(* PLC project FiveDofPlatform_v26085.modbus_registers.import.xml, CODESYS CODESYS V3.5 SP20 Patch 4 *)
(* stored: creationDateTime 2026-08-01T14:33:36, modificationDateTime 2026-08-01T14:33:36 *)

PROGRAM AxisEnableControl_PRG
  VAR
    i : INT;
    xEnableAll : BOOL;
    wEnableFeedback : WORD;
  END_VAR

            
// v26085：五轴使能寄存器 arReg_data[32] 已集中到 ModbusTcpSlave 解析。
// 本程序只保留任务调用占位，不再读写 arReg_data，避免同一个寄存器被多处写入。
          
END_PROGRAM

PROGRAM FiveDOF_Platform_PRG
  VAR
    final_angle : ARRAY[1..AXIS_COUNT] OF LREAL;  (* 最终目标 *)
    final_vel : ARRAY[1..AXIS_COUNT] OF LREAL;
    fbMove_2 : FB_5DOF_Platform_Move;  (* 功能块实例 *)
    trig_start : R_TRIG;  (* 触发边沿检测 *)
    i : INT;  (* 辅助 *)
    log_msg : STRING(255);
    logfb : Syslog_FB;
  END_VAR

            
// --------------------------------------------------
// 主逻辑
// --------------------------------------------------
// 五轴使能由 AxisEnableControl_PRG 根据 arReg_data[32] 统一控制。
// 这里不再每周期强制 TRUE，避免覆盖寄存器关闭使能命令。
// v26085：arAi_data[9] 五轴运行状态输入寄存器改由 ModbusTcpSlave 统一写出。
// 本程序只维护内部状态变量 bfiveDOF_state。
// 检测外部移动指令
trig_start(CLK := Move_5Axis_Sign=1);
IF trig_start.Q THEN

	log_msg := 'five-axis platform starts moving';
// 	logfb(write:=TRUE,sFileTestString:=log_msg);
	AppendLog(log_msg);

    // 使能所有轴（可放在这里一次性使能）
	bfiveDOF_state:=1;//开始运动
    AppendLog('status 0:6-axis start move' );
    step := 10;   // 开始安全顺序
END_IF

CASE step OF
    0: // 空闲
		bfiveDOF_state:=0;//开始运动
    // ---------- 阶段1：轴移动到目标 ----------
    10:
		FOR i := 1 TO AXIS_COUNT DO
			final_angle[i] := PlatformTargetAngle[i];
			final_vel[i]   := 360*6000/60;
			Axes[i].AxisDone := FALSE;  
			GVL.Axes[i].NeedMoveAxis := TRUE;
		END_FOR
        fbMove_2(AxisAngle := final_angle, AxisVel := final_vel, Execute := TRUE,Monitor:=TRUE);
        step := 20;

		log_msg := 'State 20: Start moving XYABC AXIS... ';
// 		logfb(write:=TRUE,sFileTestString:=log_msg);
		AppendLog(log_msg);;
    20:
        fbMove_2(AxisAngle := final_angle, AxisVel := final_vel, Execute := FALSE,Monitor:=TRUE);
        IF fbMove_2.allDone THEN
			log_msg := 'State 21: XYZABC AXIS movement completed';
// 			logfb(write:=TRUE,sFileTestString:=log_msg);
			AppendLog(log_msg);
        ELSIF fbMove_2.Error THEN
            bfiveDOF_state:=2;
        END_IF
		step := 0;

        
        
END_CASE
          
END_PROGRAM

PROGRAM AxisStatusFeedback_PRG
  VAR
    fbStatusX : Sm3_Basic.MC_ReadStatus;
    fbAxisErrorX : Sm3_Basic.MC_ReadAxisError;
    fbStatusY : Sm3_Basic.MC_ReadStatus;
    fbAxisErrorY : Sm3_Basic.MC_ReadAxisError;
    fbStatusZ : Sm3_Basic.MC_ReadStatus;
    fbAxisErrorZ : Sm3_Basic.MC_ReadAxisError;
    fbStatusB : Sm3_Basic.MC_ReadStatus;
    fbAxisErrorB : Sm3_Basic.MC_ReadAxisError;
    fbStatusC : Sm3_Basic.MC_ReadStatus;
    fbAxisErrorC : Sm3_Basic.MC_ReadAxisError;
    wStatusX : WORD;
    wStatusY : WORD;
    wStatusZ : WORD;
    wStatusB : WORD;
    wStatusC : WORD;
    dwAxisErrorX : DWORD;
    dwAxisErrorY : DWORD;
    dwAxisErrorZ : DWORD;
    dwAxisErrorB : DWORD;
    dwAxisErrorC : DWORD;
    bStatusErrorX : BOOL;
    bStatusFBErrorX : BOOL;
    bAxisErrorX : BOOL;
    bSwEndSwitchX : BOOL;
    bStatusErrorY : BOOL;
    bStatusFBErrorY : BOOL;
    bAxisErrorY : BOOL;
    bSwEndSwitchY : BOOL;
    bStatusErrorZ : BOOL;
    bStatusFBErrorZ : BOOL;
    bAxisErrorZ : BOOL;
    bSwEndSwitchZ : BOOL;
    bStatusErrorB : BOOL;
    bStatusFBErrorB : BOOL;
    bAxisErrorB : BOOL;
    bSwEndSwitchB : BOOL;
    bStatusErrorC : BOOL;
    bStatusFBErrorC : BOOL;
    bAxisErrorC : BOOL;
    bSwEndSwitchC : BOOL;
    eStatusErrorX : SMC_ERROR;
    eAxisReadErrorX : SMC_ERROR;
    bAxisReadErrorX : BOOL;
    eStatusErrorY : SMC_ERROR;
    eAxisReadErrorY : SMC_ERROR;
    bAxisReadErrorY : BOOL;
    eStatusErrorZ : SMC_ERROR;
    eAxisReadErrorZ : SMC_ERROR;
    bAxisReadErrorZ : BOOL;
    eStatusErrorB : SMC_ERROR;
    eAxisReadErrorB : SMC_ERROR;
    bAxisReadErrorB : BOOL;
    eStatusErrorC : SMC_ERROR;
    eAxisReadErrorC : SMC_ERROR;
    bAxisReadErrorC : BOOL;
    wEnableMismatchFeedback : WORD;
    wStatusErrorFeedback : WORD;
    wAxisReadErrorFeedback : WORD;
    wStatusFBErrorFeedback : WORD;
  END_VAR

            
// v26085：本程序只读取 SoftMotion 状态并写入全局缓存。
// 所有 arReg_data 寄存器地址统一在 ModbusTcpSlave 中写出，方便集中排查。

fbStatusX(
    Axis := AXIS_X,
    Enable := TRUE,
    Valid => ,
    Busy => ,
    Error => bStatusErrorX,
    ErrorID => eStatusErrorX,
    Disabled => ,
    Errorstop => ,
    Stopping => ,
    StandStill => ,
    DiscreteMotion => ,
    ContinuousMotion => ,
    SynchronizedMotion => ,
    Homing => ,
    ConstantVelocity => ,
    Accelerating => ,
    Decelerating => ,
    FBErrorOccured => bStatusFBErrorX,
);

// 读取 X 轴本体错误。这里不直接写 arReg_data，寄存器统一由 ModbusTcpSlave 输出。
fbAxisErrorX(
    Axis := AXIS_X,
    Enable := TRUE,
    Valid => ,
    Busy => ,
    Error => bAxisReadErrorX,
    ErrorID => eAxisReadErrorX,
    AxisError => bAxisErrorX,
    AxisErrorID => dwAxisErrorX,
    SWEndSwitchActive => bSwEndSwitchX
);
IF NOT bAxisErrorX THEN
    // 无轴本体错误时清零 AxisErrorID 缓存，避免保留上一次错误号。
    dwAxisErrorX := DWORD#0;
END_IF;

// 把 X 轴状态压缩成 WORD 缓存。实际 arReg_data[33] 由 ModbusTcpSlave 写出。
wStatusX := WORD#0;
IF fbStatusX.Disabled THEN wStatusX := wStatusX OR WORD#16#0001; END_IF;
IF fbStatusX.Errorstop THEN wStatusX := wStatusX OR WORD#16#0002; END_IF;
IF fbStatusX.Stopping THEN wStatusX := wStatusX OR WORD#16#0004; END_IF;
IF fbStatusX.StandStill THEN wStatusX := wStatusX OR WORD#16#0008; END_IF;
IF fbStatusX.DiscreteMotion THEN wStatusX := wStatusX OR WORD#16#0010; END_IF;
IF fbStatusX.ContinuousMotion THEN wStatusX := wStatusX OR WORD#16#0020; END_IF;
IF fbStatusX.SynchronizedMotion THEN wStatusX := wStatusX OR WORD#16#0040; END_IF;
IF fbStatusX.Homing THEN wStatusX := wStatusX OR WORD#16#0080; END_IF;
IF fbStatusX.ConstantVelocity THEN wStatusX := wStatusX OR WORD#16#0100; END_IF;
IF fbStatusX.Accelerating THEN wStatusX := wStatusX OR WORD#16#0200; END_IF;
IF fbStatusX.Decelerating THEN wStatusX := wStatusX OR WORD#16#0400; END_IF;
IF bAxisErrorX THEN wStatusX := wStatusX OR WORD#16#4000; END_IF;
IF bSwEndSwitchX THEN wStatusX := wStatusX OR WORD#16#8000; END_IF;
wAxisStatusReg[1] := wStatusX;

// 错误号先放入全局缓存，ModbusTcpSlave 统一拆成低/高 16 位寄存器。
dwAxisErrorIDReg[1] := dwAxisErrorX;
dwReadStatusErrorIDReg[1] := TO_DWORD(eStatusErrorX);
dwReadAxisErrorFBIDReg[1] := TO_DWORD(eAxisReadErrorX);

fbStatusY(
    Axis := AXIS_Y,
    Enable := TRUE,
    Valid => ,
    Busy => ,
    Error => bStatusErrorY,
    ErrorID => eStatusErrorY,
    Disabled => ,
    Errorstop => ,
    Stopping => ,
    StandStill => ,
    DiscreteMotion => ,
    ContinuousMotion => ,
    SynchronizedMotion => ,
    Homing => ,
    ConstantVelocity => ,
    Accelerating => ,
    Decelerating => ,
    FBErrorOccured => bStatusFBErrorY,
);

// 读取 Y 轴本体错误。这里不直接写 arReg_data，寄存器统一由 ModbusTcpSlave 输出。
fbAxisErrorY(
    Axis := AXIS_Y,
    Enable := TRUE,
    Valid => ,
    Busy => ,
    Error => bAxisReadErrorY,
    ErrorID => eAxisReadErrorY,
    AxisError => bAxisErrorY,
    AxisErrorID => dwAxisErrorY,
    SWEndSwitchActive => bSwEndSwitchY
);
IF NOT bAxisErrorY THEN
    // 无轴本体错误时清零 AxisErrorID 缓存，避免保留上一次错误号。
    dwAxisErrorY := DWORD#0;
END_IF;

// 把 Y 轴状态压缩成 WORD 缓存。实际 arReg_data[34] 由 ModbusTcpSlave 写出。
wStatusY := WORD#0;
IF fbStatusY.Disabled THEN wStatusY := wStatusY OR WORD#16#0001; END_IF;
IF fbStatusY.Errorstop THEN wStatusY := wStatusY OR WORD#16#0002; END_IF;
IF fbStatusY.Stopping THEN wStatusY := wStatusY OR WORD#16#0004; END_IF;
IF fbStatusY.StandStill THEN wStatusY := wStatusY OR WORD#16#0008; END_IF;
IF fbStatusY.DiscreteMotion THEN wStatusY := wStatusY OR WORD#16#0010; END_IF;
IF fbStatusY.ContinuousMotion THEN wStatusY := wStatusY OR WORD#16#0020; END_IF;
IF fbStatusY.SynchronizedMotion THEN wStatusY := wStatusY OR WORD#16#0040; END_IF;
IF fbStatusY.Homing THEN wStatusY := wStatusY OR WORD#16#0080; END_IF;
IF fbStatusY.ConstantVelocity THEN wStatusY := wStatusY OR WORD#16#0100; END_IF;
IF fbStatusY.Accelerating THEN wStatusY := wStatusY OR WORD#16#0200; END_IF;
IF fbStatusY.Decelerating THEN wStatusY := wStatusY OR WORD#16#0400; END_IF;
IF bAxisErrorY THEN wStatusY := wStatusY OR WORD#16#4000; END_IF;
IF bSwEndSwitchY THEN wStatusY := wStatusY OR WORD#16#8000; END_IF;
wAxisStatusReg[2] := wStatusY;

// 错误号先放入全局缓存，ModbusTcpSlave 统一拆成低/高 16 位寄存器。
dwAxisErrorIDReg[2] := dwAxisErrorY;
dwReadStatusErrorIDReg[2] := TO_DWORD(eStatusErrorY);
dwReadAxisErrorFBIDReg[2] := TO_DWORD(eAxisReadErrorY);

fbStatusZ(
    Axis := AXIS_Z,
    Enable := TRUE,
    Valid => ,
    Busy => ,
    Error => bStatusErrorZ,
    ErrorID => eStatusErrorZ,
    Disabled => ,
    Errorstop => ,
    Stopping => ,
    StandStill => ,
    DiscreteMotion => ,
    ContinuousMotion => ,
    SynchronizedMotion => ,
    Homing => ,
    ConstantVelocity => ,
    Accelerating => ,
    Decelerating => ,
    FBErrorOccured => bStatusFBErrorZ,
);

// 读取 Z 轴本体错误。这里不直接写 arReg_data，寄存器统一由 ModbusTcpSlave 输出。
fbAxisErrorZ(
    Axis := AXIS_Z,
    Enable := TRUE,
    Valid => ,
    Busy => ,
    Error => bAxisReadErrorZ,
    ErrorID => eAxisReadErrorZ,
    AxisError => bAxisErrorZ,
    AxisErrorID => dwAxisErrorZ,
    SWEndSwitchActive => bSwEndSwitchZ
);
IF NOT bAxisErrorZ THEN
    // 无轴本体错误时清零 AxisErrorID 缓存，避免保留上一次错误号。
    dwAxisErrorZ := DWORD#0;
END_IF;

// 把 Z 轴状态压缩成 WORD 缓存。实际 arReg_data[35] 由 ModbusTcpSlave 写出。
wStatusZ := WORD#0;
IF fbStatusZ.Disabled THEN wStatusZ := wStatusZ OR WORD#16#0001; END_IF;
IF fbStatusZ.Errorstop THEN wStatusZ := wStatusZ OR WORD#16#0002; END_IF;
IF fbStatusZ.Stopping THEN wStatusZ := wStatusZ OR WORD#16#0004; END_IF;
IF fbStatusZ.StandStill THEN wStatusZ := wStatusZ OR WORD#16#0008; END_IF;
IF fbStatusZ.DiscreteMotion THEN wStatusZ := wStatusZ OR WORD#16#0010; END_IF;
IF fbStatusZ.ContinuousMotion THEN wStatusZ := wStatusZ OR WORD#16#0020; END_IF;
IF fbStatusZ.SynchronizedMotion THEN wStatusZ := wStatusZ OR WORD#16#0040; END_IF;
IF fbStatusZ.Homing THEN wStatusZ := wStatusZ OR WORD#16#0080; END_IF;
IF fbStatusZ.ConstantVelocity THEN wStatusZ := wStatusZ OR WORD#16#0100; END_IF;
IF fbStatusZ.Accelerating THEN wStatusZ := wStatusZ OR WORD#16#0200; END_IF;
IF fbStatusZ.Decelerating THEN wStatusZ := wStatusZ OR WORD#16#0400; END_IF;
IF bAxisErrorZ THEN wStatusZ := wStatusZ OR WORD#16#4000; END_IF;
IF bSwEndSwitchZ THEN wStatusZ := wStatusZ OR WORD#16#8000; END_IF;
wAxisStatusReg[3] := wStatusZ;

// 错误号先放入全局缓存，ModbusTcpSlave 统一拆成低/高 16 位寄存器。
dwAxisErrorIDReg[3] := dwAxisErrorZ;
dwReadStatusErrorIDReg[3] := TO_DWORD(eStatusErrorZ);
dwReadAxisErrorFBIDReg[3] := TO_DWORD(eAxisReadErrorZ);

fbStatusB(
    Axis := AXIS_B,
    Enable := TRUE,
    Valid => ,
    Busy => ,
    Error => bStatusErrorB,
    ErrorID => eStatusErrorB,
    Disabled => ,
    Errorstop => ,
    Stopping => ,
    StandStill => ,
    DiscreteMotion => ,
    ContinuousMotion => ,
    SynchronizedMotion => ,
    Homing => ,
    ConstantVelocity => ,
    Accelerating => ,
    Decelerating => ,
    FBErrorOccured => bStatusFBErrorB,
);

// 读取 B 轴本体错误。这里不直接写 arReg_data，寄存器统一由 ModbusTcpSlave 输出。
fbAxisErrorB(
    Axis := AXIS_B,
    Enable := TRUE,
    Valid => ,
    Busy => ,
    Error => bAxisReadErrorB,
    ErrorID => eAxisReadErrorB,
    AxisError => bAxisErrorB,
    AxisErrorID => dwAxisErrorB,
    SWEndSwitchActive => bSwEndSwitchB
);
IF NOT bAxisErrorB THEN
    // 无轴本体错误时清零 AxisErrorID 缓存，避免保留上一次错误号。
    dwAxisErrorB := DWORD#0;
END_IF;

// 把 B 轴状态压缩成 WORD 缓存。实际 arReg_data[36] 由 ModbusTcpSlave 写出。
wStatusB := WORD#0;
IF fbStatusB.Disabled THEN wStatusB := wStatusB OR WORD#16#0001; END_IF;
IF fbStatusB.Errorstop THEN wStatusB := wStatusB OR WORD#16#0002; END_IF;
IF fbStatusB.Stopping THEN wStatusB := wStatusB OR WORD#16#0004; END_IF;
IF fbStatusB.StandStill THEN wStatusB := wStatusB OR WORD#16#0008; END_IF;
IF fbStatusB.DiscreteMotion THEN wStatusB := wStatusB OR WORD#16#0010; END_IF;
IF fbStatusB.ContinuousMotion THEN wStatusB := wStatusB OR WORD#16#0020; END_IF;
IF fbStatusB.SynchronizedMotion THEN wStatusB := wStatusB OR WORD#16#0040; END_IF;
IF fbStatusB.Homing THEN wStatusB := wStatusB OR WORD#16#0080; END_IF;
IF fbStatusB.ConstantVelocity THEN wStatusB := wStatusB OR WORD#16#0100; END_IF;
IF fbStatusB.Accelerating THEN wStatusB := wStatusB OR WORD#16#0200; END_IF;
IF fbStatusB.Decelerating THEN wStatusB := wStatusB OR WORD#16#0400; END_IF;
IF bAxisErrorB THEN wStatusB := wStatusB OR WORD#16#4000; END_IF;
IF bSwEndSwitchB THEN wStatusB := wStatusB OR WORD#16#8000; END_IF;
wAxisStatusReg[4] := wStatusB;

// 错误号先放入全局缓存，ModbusTcpSlave 统一拆成低/高 16 位寄存器。
dwAxisErrorIDReg[4] := dwAxisErrorB;
dwReadStatusErrorIDReg[4] := TO_DWORD(eStatusErrorB);
dwReadAxisErrorFBIDReg[4] := TO_DWORD(eAxisReadErrorB);

fbStatusC(
    Axis := AXIS_C,
    Enable := TRUE,
    Valid => ,
    Busy => ,
    Error => bStatusErrorC,
    ErrorID => eStatusErrorC,
    Disabled => ,
    Errorstop => ,
    Stopping => ,
    StandStill => ,
    DiscreteMotion => ,
    ContinuousMotion => ,
    SynchronizedMotion => ,
    Homing => ,
    ConstantVelocity => ,
    Accelerating => ,
    Decelerating => ,
    FBErrorOccured => bStatusFBErrorC,
);

// 读取 C 轴本体错误。这里不直接写 arReg_data，寄存器统一由 ModbusTcpSlave 输出。
fbAxisErrorC(
    Axis := AXIS_C,
    Enable := TRUE,
    Valid => ,
    Busy => ,
    Error => bAxisReadErrorC,
    ErrorID => eAxisReadErrorC,
    AxisError => bAxisErrorC,
    AxisErrorID => dwAxisErrorC,
    SWEndSwitchActive => bSwEndSwitchC
);
IF NOT bAxisErrorC THEN
    // 无轴本体错误时清零 AxisErrorID 缓存，避免保留上一次错误号。
    dwAxisErrorC := DWORD#0;
END_IF;

// 把 C 轴状态压缩成 WORD 缓存。实际 arReg_data[37] 由 ModbusTcpSlave 写出。
wStatusC := WORD#0;
IF fbStatusC.Disabled THEN wStatusC := wStatusC OR WORD#16#0001; END_IF;
IF fbStatusC.Errorstop THEN wStatusC := wStatusC OR WORD#16#0002; END_IF;
IF fbStatusC.Stopping THEN wStatusC := wStatusC OR WORD#16#0004; END_IF;
IF fbStatusC.StandStill THEN wStatusC := wStatusC OR WORD#16#0008; END_IF;
IF fbStatusC.DiscreteMotion THEN wStatusC := wStatusC OR WORD#16#0010; END_IF;
IF fbStatusC.ContinuousMotion THEN wStatusC := wStatusC OR WORD#16#0020; END_IF;
IF fbStatusC.SynchronizedMotion THEN wStatusC := wStatusC OR WORD#16#0040; END_IF;
IF fbStatusC.Homing THEN wStatusC := wStatusC OR WORD#16#0080; END_IF;
IF fbStatusC.ConstantVelocity THEN wStatusC := wStatusC OR WORD#16#0100; END_IF;
IF fbStatusC.Accelerating THEN wStatusC := wStatusC OR WORD#16#0200; END_IF;
IF fbStatusC.Decelerating THEN wStatusC := wStatusC OR WORD#16#0400; END_IF;
IF bAxisErrorC THEN wStatusC := wStatusC OR WORD#16#4000; END_IF;
IF bSwEndSwitchC THEN wStatusC := wStatusC OR WORD#16#8000; END_IF;
wAxisStatusReg[5] := wStatusC;

// 错误号先放入全局缓存，ModbusTcpSlave 统一拆成低/高 16 位寄存器。
dwAxisErrorIDReg[5] := dwAxisErrorC;
dwReadStatusErrorIDReg[5] := TO_DWORD(eStatusErrorC);
dwReadAxisErrorFBIDReg[5] := TO_DWORD(eAxisReadErrorC);

// 使能请求不一致：AxisEnable 请求 TRUE，但轴状态仍 Disabled。
wEnableMismatchFeedback := WORD#0;
IF GVL.Axes[1].AxisEnable AND fbStatusX.Disabled THEN wEnableMismatchFeedback := wEnableMismatchFeedback OR WORD#16#0001; END_IF;
IF GVL.Axes[2].AxisEnable AND fbStatusY.Disabled THEN wEnableMismatchFeedback := wEnableMismatchFeedback OR WORD#16#0002; END_IF;
IF GVL.Axes[3].AxisEnable AND fbStatusZ.Disabled THEN wEnableMismatchFeedback := wEnableMismatchFeedback OR WORD#16#0004; END_IF;
IF GVL.Axes[4].AxisEnable AND fbStatusB.Disabled THEN wEnableMismatchFeedback := wEnableMismatchFeedback OR WORD#16#0008; END_IF;
IF GVL.Axes[5].AxisEnable AND fbStatusC.Disabled THEN wEnableMismatchFeedback := wEnableMismatchFeedback OR WORD#16#0010; END_IF;
wEnableMismatchReg := wEnableMismatchFeedback;

// MC_ReadStatus.Error 汇总位，bit0..bit4=X/Y/Z/B/C。
wStatusErrorFeedback := WORD#0;
IF bStatusErrorX THEN wStatusErrorFeedback := wStatusErrorFeedback OR WORD#16#0001; END_IF;
IF bStatusErrorY THEN wStatusErrorFeedback := wStatusErrorFeedback OR WORD#16#0002; END_IF;
IF bStatusErrorZ THEN wStatusErrorFeedback := wStatusErrorFeedback OR WORD#16#0004; END_IF;
IF bStatusErrorB THEN wStatusErrorFeedback := wStatusErrorFeedback OR WORD#16#0008; END_IF;
IF bStatusErrorC THEN wStatusErrorFeedback := wStatusErrorFeedback OR WORD#16#0010; END_IF;
wReadStatusErrorBitsReg := wStatusErrorFeedback;

// MC_ReadAxisError.Error 汇总位，bit0..bit4=X/Y/Z/B/C。
wAxisReadErrorFeedback := WORD#0;
IF bAxisReadErrorX THEN wAxisReadErrorFeedback := wAxisReadErrorFeedback OR WORD#16#0001; END_IF;
IF bAxisReadErrorY THEN wAxisReadErrorFeedback := wAxisReadErrorFeedback OR WORD#16#0002; END_IF;
IF bAxisReadErrorZ THEN wAxisReadErrorFeedback := wAxisReadErrorFeedback OR WORD#16#0004; END_IF;
IF bAxisReadErrorB THEN wAxisReadErrorFeedback := wAxisReadErrorFeedback OR WORD#16#0008; END_IF;
IF bAxisReadErrorC THEN wAxisReadErrorFeedback := wAxisReadErrorFeedback OR WORD#16#0010; END_IF;
wReadAxisErrorBitsReg := wAxisReadErrorFeedback;

// MC_ReadStatus.FBErrorOccured 汇总位，bit0..bit4=X/Y/Z/B/C。
wStatusFBErrorFeedback := WORD#0;
IF bStatusFBErrorX THEN wStatusFBErrorFeedback := wStatusFBErrorFeedback OR WORD#16#0001; END_IF;
IF bStatusFBErrorY THEN wStatusFBErrorFeedback := wStatusFBErrorFeedback OR WORD#16#0002; END_IF;
IF bStatusFBErrorZ THEN wStatusFBErrorFeedback := wStatusFBErrorFeedback OR WORD#16#0004; END_IF;
IF bStatusFBErrorB THEN wStatusFBErrorFeedback := wStatusFBErrorFeedback OR WORD#16#0008; END_IF;
IF bStatusFBErrorC THEN wStatusFBErrorFeedback := wStatusFBErrorFeedback OR WORD#16#0010; END_IF;
wReadStatusFBErrorBitsReg := wStatusFBErrorFeedback;

          
END_PROGRAM

PROGRAM AXIS_X_PRG
  VAR
    伺服使能 : Sm3_Basic.MC_Power;  (* 轴功能块实例 *)
    伺服绝对位置执行 : Sm3_Basic.MC_MoveAbsolute;
    伺服实际位置 : Sm3_Basic.MC_ReadActualPosition;
    伺服停止 : Sm3_Basic.MC_Stop;
    伺服复位 : Sm3_Basic.MC_Reset;
    伺服状态 : Sm3_Basic.MC_ReadStatus;
    复位轴组 : Sm3_Basic.SMC3_ReinitDrive;
    当前位置 : LREAL;  (* 变量 *)
    轴组复位 : BOOL;
    目标位置 : LREAL;
    目标速度 : LREAL;
    伺服错误状态 : BOOL;
    轴使能状态 : BOOL;
    总线状态 : BOOL;
    复位触发 : R_TRIG;  (* 报警清除相关 *)
    复位请求 : BOOL;
    复位中 : BOOL;
    POS_DEAD_ZONE : REAL := 0.01;  (* 死区常量 *)
    move_trigger : R_TRIG;
    AXIS_X_EXCUSE : BOOL := FALSE;
    log_msg : STRING(100);
    bPowerErrorDiag : BOOL;
    ePowerErrorDiag : SMC_ERROR;
    wPowerDiag : WORD;
  END_VAR

            //------------------------------------------------------------------
// Z 轴控制逻辑（简化版 - 仅上升沿触发）
//------------------------------------------------------------------

// 读取实际位置
伺服实际位置(
    Axis    := AXIS_X,
    Enable  := TRUE,
    Position=> 当前位置
);
GVL.Axes[1].ActualAngle := 当前位置;

// 读取轴状态
伺服状态(
    Axis    := AXIS_X,
    Enable  := TRUE,
    Valid   => ,
    Busy    => ,
    Error   => 伺服错误状态,
    ErrorID => ,
    Disabled=> 总线状态
);

// 轴使能控制
伺服使能(
    Axis               := AXIS_X,
    Enable             := TRUE,
    bRegulatorOn       := GVL.Axes[1].AxisEnable,
    bDriveStart        := GVL.Axes[1].AxisEnable,
    Status             => 轴使能状态,
    bRegulatorRealState=> ,
    bDriveStartRealState=> ,
    Busy               => ,
    Error              => bPowerErrorDiag,
    ErrorID            => ePowerErrorDiag
);



// v26085：本轴 MC_Power 诊断先写入全局缓存，实际寄存器输出统一由 ModbusTcpSlave 完成。
dwPowerErrorIDReg[1] := TO_DWORD(ePowerErrorDiag);

// wPowerDiagReg[1] bit0=MC_Power.Status，bit1=MC_Power.Error。
wPowerDiag := WORD#0;
IF 轴使能状态 THEN wPowerDiag := wPowerDiag OR WORD#16#0001; END_IF;
IF bPowerErrorDiag THEN wPowerDiag := wPowerDiag OR WORD#16#0002; END_IF;
wPowerDiagReg[1] := wPowerDiag;

// 目标位置、速度赋值（来自全局变量）
目标位置 := GVL.Axes[1].TargetAngle;
目标速度 :=  GVL.Axes[1].TargetVel;

// ********** 核心：上升沿触发运动 **********
// 使用 R_TRIG 检测 need_move 的上升沿
move_trigger(CLK := GVL.Axes[1].NeedMoveAxis);
IF move_trigger.Q THEN
    AXIS_X_EXCUSE := TRUE;   // 产生一个扫描周期的脉冲
	log_msg := 'X-axis has been triggered';
// 	logfb(write:=TRUE,sFileTestString:=log_msg);
	AppendLog(log_msg);
ELSE
    AXIS_X_EXCUSE := FALSE;
END_IF

// 绝对定位指令
GVL.Axes[1].伺服绝对位置执行(
    Axis        := AXIS_X,
    Execute     := AXIS_X_EXCUSE,
    Position    := 目标位置,
    Velocity    := 目标速度,
    Acceleration:= 10000,//4000  //85000
    Deceleration:= 10000,//4000  //85000
    Jerk        := ,
    Direction   := ,
    BufferMode  := ,
    Done        => GVL.Axes[1].InitDone,
    Busy        => ,
    Active      => ,
    CommandAborted=> ,
    Error       => GVL.Axes[1].AxisError,
    ErrorID     =>
);

// 运动完成：清除 need_move 并通知状态机
IF  GVL.Axes[1].InitDone THEN
    GVL.Axes[1].NeedMoveAxis := FALSE;              // 清除运动请求
    GVL.Axes[1].AxisDone := TRUE;         // 通知状态机运动完成
	log_msg := 'X-Axis movement completed! ';
// 	logfb(write:=TRUE,sFileTestString:=log_msg);
// 	AppendLog(log_msg);
END_IF

// 复位功能块（保持不变）
伺服复位(
    Axis    := AXIS_X,
    Execute := 复位中 AND NOT 伺服复位.Done,
    Done    => ,
    Busy    => ,
    Error   => ,
    ErrorID =>
);

复位轴组(
    Axis      := AXIS_X,
    bExecute  := 伺服复位.Done,
    bVirtual  := FALSE,
    bDone     => ,
    bBusy     => ,
    bError    => ,
    nErrorID  =>
);

// 报警清除逻辑
复位触发(CLK := (伺服错误状态 OR 复位请求) AND NOT 复位中);
IF 复位触发.Q THEN
    复位中 := TRUE;
    复位请求 := FALSE;
END_IF

IF 伺服复位.Done THEN
    复位中 := FALSE;
END_IF
          
END_PROGRAM

PROGRAM Axis_Y_PRG
  VAR
    伺服使能 : Sm3_Basic.MC_Power;  (* 轴功能块实例 *)
    伺服绝对位置执行 : Sm3_Basic.MC_MoveAbsolute;
    伺服实际位置 : Sm3_Basic.MC_ReadActualPosition;
    伺服停止 : Sm3_Basic.MC_Stop;
    伺服复位 : Sm3_Basic.MC_Reset;
    伺服状态 : Sm3_Basic.MC_ReadStatus;
    复位轴组 : Sm3_Basic.SMC3_ReinitDrive;
    当前位置 : LREAL;  (* 变量 *)
    轴组复位 : BOOL;
    目标位置 : LREAL;
    目标速度 : LREAL;
    伺服错误状态 : BOOL;
    轴使能状态 : BOOL;
    总线状态 : BOOL;
    复位触发 : R_TRIG;  (* 报警清除相关 *)
    复位请求 : BOOL;
    复位中 : BOOL;
    POS_DEAD_ZONE : REAL := 0.01;  (* 死区常量 *)
    伺服复位_Done : BOOL;
    debug_Done_Status : BOOL;  (* 在 AXIS_Y0_PRG 中添加 *)
    debug_KeepEnable : BOOL;
    move_trigger : R_TRIG;  (* 脉冲触发相关 *)
    AXIS_Y_EXCUSE : BOOL := FALSE;
    log_msg : STRING(100);
    bPowerErrorDiag : BOOL;
    ePowerErrorDiag : SMC_ERROR;
    wPowerDiag : WORD;
  END_VAR

            //------------------------------------------------------------------
// Z 轴控制逻辑（简化版 - 仅上升沿触发）
//------------------------------------------------------------------

// 读取实际位置
伺服实际位置(
    Axis    := AXIS_Y,
    Enable  := TRUE,
    Position=> 当前位置
);
GVL.Axes[2].ActualAngle := 当前位置;

// 读取轴状态
伺服状态(
    Axis    := AXIS_Y,
    Enable  := TRUE,
    Valid   => ,
    Busy    => ,
    Error   => 伺服错误状态,
    ErrorID => ,
    Disabled=> 总线状态
);

// 轴使能控制
伺服使能(
    Axis               := AXIS_Y,
    Enable             := TRUE,
    bRegulatorOn       := GVL.Axes[2].AxisEnable,
    bDriveStart        := GVL.Axes[2].AxisEnable,
    Status             => 轴使能状态,
    bRegulatorRealState=> ,
    bDriveStartRealState=> ,
    Busy               => ,
    Error              => bPowerErrorDiag,
    ErrorID            => ePowerErrorDiag
);



// v26085：本轴 MC_Power 诊断先写入全局缓存，实际寄存器输出统一由 ModbusTcpSlave 完成。
dwPowerErrorIDReg[2] := TO_DWORD(ePowerErrorDiag);

// wPowerDiagReg[2] bit0=MC_Power.Status，bit1=MC_Power.Error。
wPowerDiag := WORD#0;
IF 轴使能状态 THEN wPowerDiag := wPowerDiag OR WORD#16#0001; END_IF;
IF bPowerErrorDiag THEN wPowerDiag := wPowerDiag OR WORD#16#0002; END_IF;
wPowerDiagReg[2] := wPowerDiag;

// 目标位置、速度赋值（来自全局变量）
目标位置 := GVL.Axes[2].TargetAngle;
目标速度 :=  GVL.Axes[2].TargetVel;

// ********** 核心：上升沿触发运动 **********
// 使用 R_TRIG 检测 need_move 的上升沿
move_trigger(CLK := GVL.Axes[2].NeedMoveAxis);
IF move_trigger.Q THEN
    AXIS_Y_EXCUSE := TRUE;   // 产生一个扫描周期的脉冲
	log_msg := 'X-axis has been triggered';
// 	logfb(write:=TRUE,sFileTestString:=log_msg);
	AppendLog(log_msg);
ELSE
    AXIS_Y_EXCUSE := FALSE;
END_IF

// 绝对定位指令
GVL.Axes[2].伺服绝对位置执行(
    Axis        := AXIS_Y,
    Execute     := AXIS_Y_EXCUSE,
    Position    := 目标位置,
    Velocity    := 目标速度,
    Acceleration:= 10000,//4000  //85000
    Deceleration:= 10000,//4000  //85000
    Jerk        := ,
    Direction   := ,
    BufferMode  := ,
    Done        => GVL.Axes[2].InitDone,
    Busy        => ,
    Active      => ,
    CommandAborted=> ,
    Error       => GVL.Axes[2].AxisError,
    ErrorID     =>
);

// 运动完成：清除 need_move 并通知状态机
IF  GVL.Axes[2].InitDone THEN
    GVL.Axes[2].NeedMoveAxis := FALSE;              // 清除运动请求
    GVL.Axes[2].AxisDone := TRUE;         // 通知状态机运动完成
	log_msg := 'X-Axis movement completed! ';
// 	logfb(write:=TRUE,sFileTestString:=log_msg);
// 	AppendLog(log_msg);
END_IF

// 复位功能块（保持不变）
伺服复位(
    Axis    := AXIS_Y,
    Execute := 复位中 AND NOT 伺服复位.Done,
    Done    => ,
    Busy    => ,
    Error   => ,
    ErrorID =>
);

复位轴组(
    Axis      := AXIS_Y,
    bExecute  := 伺服复位.Done,
    bVirtual  := FALSE,
    bDone     => ,
    bBusy     => ,
    bError    => ,
    nErrorID  =>
);

// 报警清除逻辑
复位触发(CLK := (伺服错误状态 OR 复位请求) AND NOT 复位中);
IF 复位触发.Q THEN
    复位中 := TRUE;
    复位请求 := FALSE;
END_IF

IF 伺服复位.Done THEN
    复位中 := FALSE;
END_IF
          
END_PROGRAM

PROGRAM AXIS_Z_PRG
  VAR
    伺服使能 : Sm3_Basic.MC_Power;  (* 轴功能块实例 *)
    伺服绝对位置执行 : Sm3_Basic.MC_MoveAbsolute;
    伺服实际位置 : Sm3_Basic.MC_ReadActualPosition;
    伺服停止 : Sm3_Basic.MC_Stop;
    伺服复位 : Sm3_Basic.MC_Reset;
    伺服状态 : Sm3_Basic.MC_ReadStatus;
    复位轴组 : Sm3_Basic.SMC3_ReinitDrive;
    当前位置 : LREAL;  (* 变量 *)
    轴组复位 : BOOL;
    目标位置 : LREAL;
    目标速度 : LREAL;
    伺服错误状态 : BOOL;
    轴使能状态 : BOOL;
    总线状态 : BOOL;
    复位触发 : R_TRIG;  (* 报警清除相关 *)
    复位请求 : BOOL;
    复位中 : BOOL;
    伺服复位_Done : BOOL;
    debug_Done_Status : BOOL;  (* 在 AXIS_Z_PRG 中添加 *)
    debug_KeepEnable : BOOL;
    move_trigger : R_TRIG;  (* 脉冲触发相关 *)
    AXIS_Z_EXCUSE : BOOL := FALSE;
    log_msg : STRING(100);
    bPowerErrorDiag : BOOL;
    ePowerErrorDiag : SMC_ERROR;
    wPowerDiag : WORD;
  END_VAR

            //------------------------------------------------------------------
// Z 轴控制逻辑（简化版 - 仅上升沿触发）
//------------------------------------------------------------------

// 读取实际位置
伺服实际位置(
    Axis    := AXIS_Z,
    Enable  := TRUE,
    Position=> 当前位置
);
GVL.Axes[3].ActualAngle := 当前位置;

// 读取轴状态
伺服状态(
    Axis    := AXIS_Z,
    Enable  := TRUE,
    Valid   => ,
    Busy    => ,
    Error   => 伺服错误状态,
    ErrorID => ,
    Disabled=> 总线状态
);

// 轴使能控制
伺服使能(
    Axis               := AXIS_Z,
    Enable             := TRUE,
    bRegulatorOn       := GVL.Axes[3].AxisEnable,
    bDriveStart        := GVL.Axes[3].AxisEnable,
    Status             => 轴使能状态,
    bRegulatorRealState=> ,
    bDriveStartRealState=> ,
    Busy               => ,
    Error              => bPowerErrorDiag,
    ErrorID            => ePowerErrorDiag
);



// v26085：本轴 MC_Power 诊断先写入全局缓存，实际寄存器输出统一由 ModbusTcpSlave 完成。
dwPowerErrorIDReg[3] := TO_DWORD(ePowerErrorDiag);

// wPowerDiagReg[3] bit0=MC_Power.Status，bit1=MC_Power.Error。
wPowerDiag := WORD#0;
IF 轴使能状态 THEN wPowerDiag := wPowerDiag OR WORD#16#0001; END_IF;
IF bPowerErrorDiag THEN wPowerDiag := wPowerDiag OR WORD#16#0002; END_IF;
wPowerDiagReg[3] := wPowerDiag;

// 目标位置、速度赋值（来自全局变量）
目标位置 := GVL.Axes[3].TargetAngle;
目标速度 :=  GVL.Axes[3].TargetVel;

// ********** 核心：上升沿触发运动 **********
// 使用 R_TRIG 检测 need_move 的上升沿
move_trigger(CLK := GVL.Axes[3].NeedMoveAxis);
IF move_trigger.Q THEN
    AXIS_Z_EXCUSE := TRUE;   // 产生一个扫描周期的脉冲
	log_msg := 'X-axis has been triggered';
// 	logfb(write:=TRUE,sFileTestString:=log_msg);
	AppendLog(log_msg);
ELSE
    AXIS_Z_EXCUSE := FALSE;
END_IF

// 绝对定位指令
GVL.Axes[3].伺服绝对位置执行(
    Axis        := AXIS_Z,
    Execute     := AXIS_Z_EXCUSE,
    Position    := 目标位置,
    Velocity    := 目标速度,
    Acceleration:= 10000,//4000  //85000
    Deceleration:= 10000,//4000  //85000
    Jerk        := ,
    Direction   := ,
    BufferMode  := ,
    Done        => GVL.Axes[3].InitDone,
    Busy        => ,
    Active      => ,
    CommandAborted=> ,
    Error       => GVL.Axes[3].AxisError,
    ErrorID     =>
);

// 运动完成：清除 need_move 并通知状态机
IF  GVL.Axes[3].InitDone THEN
    GVL.Axes[3].NeedMoveAxis := FALSE;              // 清除运动请求
    GVL.Axes[3].AxisDone := TRUE;         // 通知状态机运动完成
	log_msg := 'Z-Axis movement completed! ';
// 	logfb(write:=TRUE,sFileTestString:=log_msg);
// 	AppendLog(log_msg);
END_IF

// 复位功能块（保持不变）
伺服复位(
    Axis    := AXIS_Z,
    Execute := 复位中 AND NOT 伺服复位.Done,
    Done    => ,
    Busy    => ,
    Error   => ,
    ErrorID =>
);

复位轴组(
    Axis      := AXIS_Z,
    bExecute  := 伺服复位.Done,
    bVirtual  := FALSE,
    bDone     => ,
    bBusy     => ,
    bError    => ,
    nErrorID  =>
);

// 报警清除逻辑
复位触发(CLK := (伺服错误状态 OR 复位请求) AND NOT 复位中);
IF 复位触发.Q THEN
    复位中 := TRUE;
    复位请求 := FALSE;
END_IF

IF 伺服复位.Done THEN
    复位中 := FALSE;
END_IF
          
END_PROGRAM

PROGRAM AXIS_B_PRG
  VAR
    伺服使能 : Sm3_Basic.MC_Power;  (* 轴功能块实例 *)
    伺服绝对位置执行 : Sm3_Basic.MC_MoveAbsolute;
    伺服实际位置 : Sm3_Basic.MC_ReadActualPosition;
    伺服停止 : Sm3_Basic.MC_Stop;
    伺服复位 : Sm3_Basic.MC_Reset;
    伺服状态 : Sm3_Basic.MC_ReadStatus;
    复位轴组 : Sm3_Basic.SMC3_ReinitDrive;
    当前位置 : LREAL;  (* 变量 *)
    轴组复位 : BOOL;
    目标位置 : LREAL;
    目标速度 : LREAL;
    伺服错误状态 : BOOL;
    轴使能状态 : BOOL;
    总线状态 : BOOL;
    复位触发 : R_TRIG;  (* 报警清除相关 *)
    复位请求 : BOOL;
    复位中 : BOOL;
    move_trigger : R_TRIG;
    AXIS_B_EXCUSE : BOOL := FALSE;
    log_msg : STRING(100);
    bPowerErrorDiag : BOOL;
    ePowerErrorDiag : SMC_ERROR;
    wPowerDiag : WORD;
  END_VAR

            //------------------------------------------------------------------
// Z 轴控制逻辑（简化版 - 仅上升沿触发）
//------------------------------------------------------------------

// 读取实际位置
伺服实际位置(
    Axis    := AXIS_B,
    Enable  := TRUE,
    Position=> 当前位置
);
GVL.Axes[4].ActualAngle := 当前位置;

// 读取轴状态
伺服状态(
    Axis    := AXIS_B,
    Enable  := TRUE,
    Valid   => ,
    Busy    => ,
    Error   => 伺服错误状态,
    ErrorID => ,
    Disabled=> 总线状态
);

// 轴使能控制
伺服使能(
    Axis               := AXIS_B,
    Enable             := TRUE,
    bRegulatorOn       := GVL.Axes[4].AxisEnable,
    bDriveStart        := GVL.Axes[4].AxisEnable,
    Status             => 轴使能状态,
    bRegulatorRealState=> ,
    bDriveStartRealState=> ,
    Busy               => ,
    Error              => bPowerErrorDiag,
    ErrorID            => ePowerErrorDiag
);



// v26085：本轴 MC_Power 诊断先写入全局缓存，实际寄存器输出统一由 ModbusTcpSlave 完成。
dwPowerErrorIDReg[4] := TO_DWORD(ePowerErrorDiag);

// wPowerDiagReg[4] bit0=MC_Power.Status，bit1=MC_Power.Error。
wPowerDiag := WORD#0;
IF 轴使能状态 THEN wPowerDiag := wPowerDiag OR WORD#16#0001; END_IF;
IF bPowerErrorDiag THEN wPowerDiag := wPowerDiag OR WORD#16#0002; END_IF;
wPowerDiagReg[4] := wPowerDiag;

// 目标位置、速度赋值（来自全局变量）
目标位置 := GVL.Axes[4].TargetAngle;
目标速度 :=  GVL.Axes[4].TargetVel;

// ********** 核心：上升沿触发运动 **********
// 使用 R_TRIG 检测 need_move 的上升沿
move_trigger(CLK := GVL.Axes[4].NeedMoveAxis);
IF move_trigger.Q THEN
    AXIS_B_EXCUSE := TRUE;   // 产生一个扫描周期的脉冲
	log_msg := 'X-axis has been triggered';
// 	logfb(write:=TRUE,sFileTestString:=log_msg);
	AppendLog(log_msg);
ELSE
    AXIS_B_EXCUSE := FALSE;
END_IF

// 绝对定位指令
GVL.Axes[4].伺服绝对位置执行(
    Axis        := AXIS_B,
    Execute     := AXIS_B_EXCUSE,
    Position    := 目标位置,
    Velocity    := 目标速度,
    Acceleration:= 10000,//4000  //85000
    Deceleration:= 10000,//4000  //85000
    Jerk        := ,
    Direction   := ,
    BufferMode  := ,
    Done        => GVL.Axes[4].InitDone,
    Busy        => ,
    Active      => ,
    CommandAborted=> ,
    Error       => GVL.Axes[4].AxisError,
    ErrorID     =>
);

// 运动完成：清除 need_move 并通知状态机
IF  GVL.Axes[4].InitDone THEN
    GVL.Axes[4].NeedMoveAxis := FALSE;              // 清除运动请求
    GVL.Axes[4].AxisDone := TRUE;         // 通知状态机运动完成
	log_msg := 'B-Axis movement completed! ';
// 	logfb(write:=TRUE,sFileTestString:=log_msg);
// 	AppendLog(log_msg);
END_IF

// 复位功能块（保持不变）
伺服复位(
    Axis    := AXIS_B,
    Execute := 复位中 AND NOT 伺服复位.Done,
    Done    => ,
    Busy    => ,
    Error   => ,
    ErrorID =>
);

复位轴组(
    Axis      := AXIS_B,
    bExecute  := 伺服复位.Done,
    bVirtual  := FALSE,
    bDone     => ,
    bBusy     => ,
    bError    => ,
    nErrorID  =>
);

// 报警清除逻辑
复位触发(CLK := (伺服错误状态 OR 复位请求) AND NOT 复位中);
IF 复位触发.Q THEN
    复位中 := TRUE;
    复位请求 := FALSE;
END_IF

IF 伺服复位.Done THEN
    复位中 := FALSE;
END_IF
          
END_PROGRAM

PROGRAM AXIS_C_PRG
  VAR
    伺服使能 : Sm3_Basic.MC_Power;  (* 轴功能块实例 *)
    伺服绝对位置执行 : Sm3_Basic.MC_MoveAbsolute;
    伺服实际位置 : Sm3_Basic.MC_ReadActualPosition;
    伺服停止 : Sm3_Basic.MC_Stop;
    伺服复位 : Sm3_Basic.MC_Reset;
    伺服状态 : Sm3_Basic.MC_ReadStatus;
    复位轴组 : Sm3_Basic.SMC3_ReinitDrive;
    当前位置 : LREAL;  (* 变量 *)
    轴组复位 : BOOL;
    目标位置 : LREAL;
    目标速度 : LREAL;
    伺服错误状态 : BOOL;
    轴使能状态 : BOOL;
    总线状态 : BOOL;
    复位触发 : R_TRIG;  (* 报警清除相关 *)
    复位请求 : BOOL;
    复位中 : BOOL;
    POS_DEAD_ZONE : REAL := 0.01;  (* 死区常量 *)
    diff_old : BOOL := FALSE;  (* 上升沿检测 *)
    diff : BOOL;
    保持使能 : BOOL := FALSE;  (* 控制 MC_Power.Enable *)
    EnRise : R_TRIG;  (* 外部使能上升沿 *)
    PowerStatusRise : R_TRIG;  (* 轴使能状态上升沿 *)
    move_trigger : R_TRIG;
    AXIS_C_EXCUSE : BOOL := FALSE;
    AXIS_C_Done_Internal : BOOL;
    log_msg : STRING(100);
    bPowerErrorDiag : BOOL;
    ePowerErrorDiag : SMC_ERROR;
    wPowerDiag : WORD;
  END_VAR

            //------------------------------------------------------------------
// Z 轴控制逻辑（简化版 - 仅上升沿触发）
//------------------------------------------------------------------

// 读取实际位置
伺服实际位置(
    Axis    := AXIS_C,
    Enable  := TRUE,
    Position=> 当前位置
);
GVL.Axes[5].ActualAngle := 当前位置;

// 读取轴状态
伺服状态(
    Axis    := AXIS_C,
    Enable  := TRUE,
    Valid   => ,
    Busy    => ,
    Error   => 伺服错误状态,
    ErrorID => ,
    Disabled=> 总线状态
);

// 轴使能控制
伺服使能(
    Axis               := AXIS_C,
    Enable             := TRUE,
    bRegulatorOn       := GVL.Axes[5].AxisEnable,
    bDriveStart        := GVL.Axes[5].AxisEnable,
    Status             => 轴使能状态,
    bRegulatorRealState=> ,
    bDriveStartRealState=> ,
    Busy               => ,
    Error              => bPowerErrorDiag,
    ErrorID            => ePowerErrorDiag
);



// v26085：本轴 MC_Power 诊断先写入全局缓存，实际寄存器输出统一由 ModbusTcpSlave 完成。
dwPowerErrorIDReg[5] := TO_DWORD(ePowerErrorDiag);

// wPowerDiagReg[5] bit0=MC_Power.Status，bit1=MC_Power.Error。
wPowerDiag := WORD#0;
IF 轴使能状态 THEN wPowerDiag := wPowerDiag OR WORD#16#0001; END_IF;
IF bPowerErrorDiag THEN wPowerDiag := wPowerDiag OR WORD#16#0002; END_IF;
wPowerDiagReg[5] := wPowerDiag;

// 目标位置、速度赋值（来自全局变量）
目标位置 := GVL.Axes[5].TargetAngle;
目标速度 :=  GVL.Axes[5].TargetVel;

// ********** 核心：上升沿触发运动 **********
// 使用 R_TRIG 检测 need_move 的上升沿
move_trigger(CLK := GVL.Axes[5].NeedMoveAxis);
IF move_trigger.Q THEN
    AXIS_C_EXCUSE := TRUE;   // 产生一个扫描周期的脉冲
	log_msg := 'C-axis has been triggered';
// 	logfb(write:=TRUE,sFileTestString:=log_msg);
	AppendLog(log_msg);
ELSE
    AXIS_C_EXCUSE := FALSE;
END_IF

// 绝对定位指令
GVL.Axes[5].伺服绝对位置执行(
    Axis        := AXIS_C,
    Execute     := AXIS_C_EXCUSE,
    Position    := 目标位置,
    Velocity    := 目标速度,
    Acceleration:= 10000,//4000  //85000
    Deceleration:= 10000,//4000  //85000
    Jerk        := ,
    Direction   := ,
    BufferMode  := ,
    Done        => GVL.Axes[5].InitDone,
    Busy        => ,
    Active      => ,
    CommandAborted=> ,
    Error       => GVL.Axes[5].AxisError,
    ErrorID     =>
);

// 运动完成：清除 need_move 并通知状态机
IF  GVL.Axes[5].InitDone THEN
    GVL.Axes[5].NeedMoveAxis := FALSE;              // 清除运动请求
    GVL.Axes[5].AxisDone := TRUE;         // 通知状态机运动完成
	log_msg := 'B-Axis movement completed! ';
// 	logfb(write:=TRUE,sFileTestString:=log_msg);
// 	AppendLog(log_msg);
END_IF

// 复位功能块（保持不变）
伺服复位(
    Axis    := AXIS_C,
    Execute := 复位中 AND NOT 伺服复位.Done,
    Done    => ,
    Busy    => ,
    Error   => ,
    ErrorID =>
);

复位轴组(
    Axis      := AXIS_C,
    bExecute  := 伺服复位.Done,
    bVirtual  := FALSE,
    bDone     => ,
    bBusy     => ,
    bError    => ,
    nErrorID  =>
);

// 报警清除逻辑
复位触发(CLK := (伺服错误状态 OR 复位请求) AND NOT 复位中);
IF 复位触发.Q THEN
    复位中 := TRUE;
    复位请求 := FALSE;
END_IF

IF 伺服复位.Done THEN
    复位中 := FALSE;
END_IF
          
END_PROGRAM

PROGRAM JogX
  VAR
    fbJogX : FB_ServoJog;
    xServoEnable : BOOL := TRUE;
    xResetCmdReg : BOOL;
  END_VAR

            
// ================================
  // 5轴点动控制
  // ================================

  // 五轴总关闭时，点动功能块不会继续用本地 TRUE 保持上使能。

  // v26085：复位命令由 ModbusTcpSlave 从 arReg_data[89] 解析到 xJogReset[1]。
  // FB_ServoJog 内部用 R_TRIG 把这个 BOOL 转成 MC_Reset 上升沿。
  xResetCmdReg := xJogReset[1];

  xServoEnable := GVL.Axes[1].AxisEnable;

  fbJogX(
      Axis := AXIS_X,
      xServoOn := xServoEnable,
      xReset := xResetCmdReg,
      xJogFwd := xJogFwd[1],
      xJogRev := xJogRev[1],
      xLimitFwd := FALSE,
      xLimitRev := FALSE,
      lrJogVel := 100.0,
      lrAcc := 100.0,
      lrDec := 200.0,
      lrJerk := 0.0
  );


  // v26085：Jog 程序只写全局反馈位图，寄存器 arReg_data[90..99] 统一由 ModbusTcpSlave 写出。
  IF xResetCmdReg THEN
    wJogResetCmdReg := wJogResetCmdReg OR WORD#16#0001;
ELSE
    wJogResetCmdReg := wJogResetCmdReg AND WORD#16#FFFE;
END_IF;
  IF xJogMode[1] THEN
    wJogModeReg := wJogModeReg OR WORD#16#0001;
ELSE
    wJogModeReg := wJogModeReg AND WORD#16#FFFE;
END_IF;
  IF xJogFwd[1] THEN
    wJogFwdReg := wJogFwdReg OR WORD#16#0001;
ELSE
    wJogFwdReg := wJogFwdReg AND WORD#16#FFFE;
END_IF;
  IF xJogRev[1] THEN
    wJogRevReg := wJogRevReg OR WORD#16#0001;
ELSE
    wJogRevReg := wJogRevReg AND WORD#16#FFFE;
END_IF;
  IF fbJogX.xReady THEN
    wJogReadyReg := wJogReadyReg OR WORD#16#0001;
ELSE
    wJogReadyReg := wJogReadyReg AND WORD#16#FFFE;
END_IF;
  IF fbJogX.xMoving THEN
    wJogMovingReg := wJogMovingReg OR WORD#16#0001;
ELSE
    wJogMovingReg := wJogMovingReg AND WORD#16#FFFE;
END_IF;
  IF fbJogX.xFault THEN
    wJogFaultReg := wJogFaultReg OR WORD#16#0001;
ELSE
    wJogFaultReg := wJogFaultReg AND WORD#16#FFFE;
END_IF;
  IF fbJogX.xJogError THEN
    wJogErrorReg := wJogErrorReg OR WORD#16#0001;
ELSE
    wJogErrorReg := wJogErrorReg AND WORD#16#FFFE;
END_IF;
  IF fbJogX.xJogAborted THEN
    wJogAbortedReg := wJogAbortedReg OR WORD#16#0001;
ELSE
    wJogAbortedReg := wJogAbortedReg AND WORD#16#FFFE;
END_IF;

          
END_PROGRAM

PROGRAM JogY
  VAR
    fbJogX : FB_ServoJog;
    fbJogY : FB_ServoJog;
    fbJogZ : FB_ServoJog;
    fbJogB : FB_ServoJog;
    fbJogC : FB_ServoJog;
    xServoEnable : BOOL := TRUE;
    xResetCmdReg : BOOL;
  END_VAR

            
// ================================
  // 5轴点动控制
  // ================================


  // 五轴总关闭时，点动功能块不会继续用本地 TRUE 保持上使能。

  // v26085：复位命令由 ModbusTcpSlave 从 arReg_data[89] 解析到 xJogReset[2]。
  // FB_ServoJog 内部用 R_TRIG 把这个 BOOL 转成 MC_Reset 上升沿。
  xResetCmdReg := xJogReset[2];

  xServoEnable := GVL.Axes[2].AxisEnable;

  fbJogY(
      Axis := AXIS_Y,
      xServoOn := xServoEnable,
      xReset := xResetCmdReg,
      xJogFwd := xJogFwd[2],
      xJogRev := xJogRev[2],
      xLimitFwd := FALSE,
      xLimitRev := FALSE,
      lrJogVel := 100.0,
      lrAcc := 100.0,
      lrDec := 200.0,
      lrJerk := 0.0
  );


  // v26085：Jog 程序只写全局反馈位图，寄存器 arReg_data[90..99] 统一由 ModbusTcpSlave 写出。
  IF xResetCmdReg THEN
    wJogResetCmdReg := wJogResetCmdReg OR WORD#16#0002;
ELSE
    wJogResetCmdReg := wJogResetCmdReg AND WORD#16#FFFD;
END_IF;
  IF xJogMode[2] THEN
    wJogModeReg := wJogModeReg OR WORD#16#0002;
ELSE
    wJogModeReg := wJogModeReg AND WORD#16#FFFD;
END_IF;
  IF xJogFwd[2] THEN
    wJogFwdReg := wJogFwdReg OR WORD#16#0002;
ELSE
    wJogFwdReg := wJogFwdReg AND WORD#16#FFFD;
END_IF;
  IF xJogRev[2] THEN
    wJogRevReg := wJogRevReg OR WORD#16#0002;
ELSE
    wJogRevReg := wJogRevReg AND WORD#16#FFFD;
END_IF;
  IF fbJogY.xReady THEN
    wJogReadyReg := wJogReadyReg OR WORD#16#0002;
ELSE
    wJogReadyReg := wJogReadyReg AND WORD#16#FFFD;
END_IF;
  IF fbJogY.xMoving THEN
    wJogMovingReg := wJogMovingReg OR WORD#16#0002;
ELSE
    wJogMovingReg := wJogMovingReg AND WORD#16#FFFD;
END_IF;
  IF fbJogY.xFault THEN
    wJogFaultReg := wJogFaultReg OR WORD#16#0002;
ELSE
    wJogFaultReg := wJogFaultReg AND WORD#16#FFFD;
END_IF;
  IF fbJogY.xJogError THEN
    wJogErrorReg := wJogErrorReg OR WORD#16#0002;
ELSE
    wJogErrorReg := wJogErrorReg AND WORD#16#FFFD;
END_IF;
  IF fbJogY.xJogAborted THEN
    wJogAbortedReg := wJogAbortedReg OR WORD#16#0002;
ELSE
    wJogAbortedReg := wJogAbortedReg AND WORD#16#FFFD;
END_IF;

          
END_PROGRAM

PROGRAM JogZ
  VAR
    fbJogX : FB_ServoJog;
    fbJogY : FB_ServoJog;
    fbJogZ : FB_ServoJog;
    fbJogB : FB_ServoJog;
    fbJogC : FB_ServoJog;
    xServoEnable : BOOL := TRUE;
    xResetCmdReg : BOOL;
  END_VAR

            
// ================================
  // 5轴点动控制
  // ================================

  

  // 五轴总关闭时，点动功能块不会继续用本地 TRUE 保持上使能。

  // v26085：复位命令由 ModbusTcpSlave 从 arReg_data[89] 解析到 xJogReset[3]。
  // FB_ServoJog 内部用 R_TRIG 把这个 BOOL 转成 MC_Reset 上升沿。
  xResetCmdReg := xJogReset[3];

  xServoEnable := GVL.Axes[3].AxisEnable;

  fbJogZ(
      Axis := AXIS_Z,
      xServoOn := xServoEnable,
      xReset := xResetCmdReg,
      xJogFwd := xJogFwd[3],
      xJogRev := xJogRev[3],
      xLimitFwd := FALSE,
      xLimitRev := FALSE,
      lrJogVel := 100.0,
      lrAcc := 100.0,
      lrDec := 200.0,
      lrJerk := 0.0
  );


  // v26085：Jog 程序只写全局反馈位图，寄存器 arReg_data[90..99] 统一由 ModbusTcpSlave 写出。
  IF xResetCmdReg THEN
    wJogResetCmdReg := wJogResetCmdReg OR WORD#16#0004;
ELSE
    wJogResetCmdReg := wJogResetCmdReg AND WORD#16#FFFB;
END_IF;
  IF xJogMode[3] THEN
    wJogModeReg := wJogModeReg OR WORD#16#0004;
ELSE
    wJogModeReg := wJogModeReg AND WORD#16#FFFB;
END_IF;
  IF xJogFwd[3] THEN
    wJogFwdReg := wJogFwdReg OR WORD#16#0004;
ELSE
    wJogFwdReg := wJogFwdReg AND WORD#16#FFFB;
END_IF;
  IF xJogRev[3] THEN
    wJogRevReg := wJogRevReg OR WORD#16#0004;
ELSE
    wJogRevReg := wJogRevReg AND WORD#16#FFFB;
END_IF;
  IF fbJogZ.xReady THEN
    wJogReadyReg := wJogReadyReg OR WORD#16#0004;
ELSE
    wJogReadyReg := wJogReadyReg AND WORD#16#FFFB;
END_IF;
  IF fbJogZ.xMoving THEN
    wJogMovingReg := wJogMovingReg OR WORD#16#0004;
ELSE
    wJogMovingReg := wJogMovingReg AND WORD#16#FFFB;
END_IF;
  IF fbJogZ.xFault THEN
    wJogFaultReg := wJogFaultReg OR WORD#16#0004;
ELSE
    wJogFaultReg := wJogFaultReg AND WORD#16#FFFB;
END_IF;
  IF fbJogZ.xJogError THEN
    wJogErrorReg := wJogErrorReg OR WORD#16#0004;
ELSE
    wJogErrorReg := wJogErrorReg AND WORD#16#FFFB;
END_IF;
  IF fbJogZ.xJogAborted THEN
    wJogAbortedReg := wJogAbortedReg OR WORD#16#0004;
ELSE
    wJogAbortedReg := wJogAbortedReg AND WORD#16#FFFB;
END_IF;

          
END_PROGRAM

PROGRAM JogB
  VAR
    fbJogX : FB_ServoJog;
    fbJogY : FB_ServoJog;
    fbJogZ : FB_ServoJog;
    fbJogB : FB_ServoJog;
    fbJogC : FB_ServoJog;
    xServoEnable : BOOL := TRUE;
    xResetCmdReg : BOOL;
  END_VAR

            
// ================================
  // 5轴点动控制
  // ================================

  
  // 五轴总关闭时，点动功能块不会继续用本地 TRUE 保持上使能。

  // v26085：复位命令由 ModbusTcpSlave 从 arReg_data[89] 解析到 xJogReset[4]。
  // FB_ServoJog 内部用 R_TRIG 把这个 BOOL 转成 MC_Reset 上升沿。
  xResetCmdReg := xJogReset[4];

  xServoEnable := GVL.Axes[4].AxisEnable;

  fbJogB(
      Axis := AXIS_B,
      xServoOn := xServoEnable,
      xReset := xResetCmdReg,
      xJogFwd := xJogFwd[4],
      xJogRev := xJogRev[4],
      xLimitFwd := FALSE,
      xLimitRev := FALSE,
      lrJogVel := 100.0,
      lrAcc := 100.0,
      lrDec := 200.0,
      lrJerk := 0.0
  );


  // v26085：Jog 程序只写全局反馈位图，寄存器 arReg_data[90..99] 统一由 ModbusTcpSlave 写出。
  IF xResetCmdReg THEN
    wJogResetCmdReg := wJogResetCmdReg OR WORD#16#0008;
ELSE
    wJogResetCmdReg := wJogResetCmdReg AND WORD#16#FFF7;
END_IF;
  IF xJogMode[4] THEN
    wJogModeReg := wJogModeReg OR WORD#16#0008;
ELSE
    wJogModeReg := wJogModeReg AND WORD#16#FFF7;
END_IF;
  IF xJogFwd[4] THEN
    wJogFwdReg := wJogFwdReg OR WORD#16#0008;
ELSE
    wJogFwdReg := wJogFwdReg AND WORD#16#FFF7;
END_IF;
  IF xJogRev[4] THEN
    wJogRevReg := wJogRevReg OR WORD#16#0008;
ELSE
    wJogRevReg := wJogRevReg AND WORD#16#FFF7;
END_IF;
  IF fbJogB.xReady THEN
    wJogReadyReg := wJogReadyReg OR WORD#16#0008;
ELSE
    wJogReadyReg := wJogReadyReg AND WORD#16#FFF7;
END_IF;
  IF fbJogB.xMoving THEN
    wJogMovingReg := wJogMovingReg OR WORD#16#0008;
ELSE
    wJogMovingReg := wJogMovingReg AND WORD#16#FFF7;
END_IF;
  IF fbJogB.xFault THEN
    wJogFaultReg := wJogFaultReg OR WORD#16#0008;
ELSE
    wJogFaultReg := wJogFaultReg AND WORD#16#FFF7;
END_IF;
  IF fbJogB.xJogError THEN
    wJogErrorReg := wJogErrorReg OR WORD#16#0008;
ELSE
    wJogErrorReg := wJogErrorReg AND WORD#16#FFF7;
END_IF;
  IF fbJogB.xJogAborted THEN
    wJogAbortedReg := wJogAbortedReg OR WORD#16#0008;
ELSE
    wJogAbortedReg := wJogAbortedReg AND WORD#16#FFF7;
END_IF;

          
END_PROGRAM

PROGRAM JogC
  VAR
    fbJogX : FB_ServoJog;
    fbJogY : FB_ServoJog;
    fbJogZ : FB_ServoJog;
    fbJogB : FB_ServoJog;
    fbJogC : FB_ServoJog;
    xServoEnable : BOOL := TRUE;
    xResetCmdReg : BOOL;
  END_VAR

            
// ================================
  // 5轴点动控制
  // ================================

  // 五轴总关闭时，点动功能块不会继续用本地 TRUE 保持上使能。

  // v26085：复位命令由 ModbusTcpSlave 从 arReg_data[89] 解析到 xJogReset[5]。
  // FB_ServoJog 内部用 R_TRIG 把这个 BOOL 转成 MC_Reset 上升沿。
  xResetCmdReg := xJogReset[5];

  xServoEnable := GVL.Axes[5].AxisEnable;

  fbJogC(
      Axis := AXIS_C,
      xServoOn := xServoEnable,
      xReset := xResetCmdReg,
      xJogFwd := xJogFwd[5],
      xJogRev := xJogRev[5],
      xLimitFwd := FALSE,
      xLimitRev := FALSE,
      lrJogVel := 100.0,
      lrAcc := 100.0,
      lrDec := 200.0,
      lrJerk := 0.0
  );


  // v26085：Jog 程序只写全局反馈位图，寄存器 arReg_data[90..99] 统一由 ModbusTcpSlave 写出。
  IF xResetCmdReg THEN
    wJogResetCmdReg := wJogResetCmdReg OR WORD#16#0010;
ELSE
    wJogResetCmdReg := wJogResetCmdReg AND WORD#16#FFEF;
END_IF;
  IF xJogMode[5] THEN
    wJogModeReg := wJogModeReg OR WORD#16#0010;
ELSE
    wJogModeReg := wJogModeReg AND WORD#16#FFEF;
END_IF;
  IF xJogFwd[5] THEN
    wJogFwdReg := wJogFwdReg OR WORD#16#0010;
ELSE
    wJogFwdReg := wJogFwdReg AND WORD#16#FFEF;
END_IF;
  IF xJogRev[5] THEN
    wJogRevReg := wJogRevReg OR WORD#16#0010;
ELSE
    wJogRevReg := wJogRevReg AND WORD#16#FFEF;
END_IF;
  IF fbJogC.xReady THEN
    wJogReadyReg := wJogReadyReg OR WORD#16#0010;
ELSE
    wJogReadyReg := wJogReadyReg AND WORD#16#FFEF;
END_IF;
  IF fbJogC.xMoving THEN
    wJogMovingReg := wJogMovingReg OR WORD#16#0010;
ELSE
    wJogMovingReg := wJogMovingReg AND WORD#16#FFEF;
END_IF;
  IF fbJogC.xFault THEN
    wJogFaultReg := wJogFaultReg OR WORD#16#0010;
ELSE
    wJogFaultReg := wJogFaultReg AND WORD#16#FFEF;
END_IF;
  IF fbJogC.xJogError THEN
    wJogErrorReg := wJogErrorReg OR WORD#16#0010;
ELSE
    wJogErrorReg := wJogErrorReg AND WORD#16#FFEF;
END_IF;
  IF fbJogC.xJogAborted THEN
    wJogAbortedReg := wJogAbortedReg OR WORD#16#0010;
ELSE
    wJogAbortedReg := wJogAbortedReg AND WORD#16#FFEF;
END_IF;

          
END_PROGRAM

PROGRAM ModbusTcpSlave
  VAR CONSTANT
    aAngleFactor : ARRAY[1..GVL.AXIS_COUNT] OF REAL := [(360.0 / 26.0), (360.0 / 5.0), (360.0 / 5.0), 1, 1];
    xEnableAllReg : BOOL;
  END_VAR
  VAR
    modTcpSlaveInit : gcan.FB_ModbusTCP_Slave_Init;  (* Modbus TCP Slave初始化功能块 *)
    modTcpSlaveCtrl : gcan.FB_ModbusTCP_Slave_Ctrl;  (* Modbus TCP Slave执行功能块 *)
    eout : BOOL;  (* 用于承接功能块中完成标志引脚数据的变量 *)
    iSocket : INT;  (* 用于存放自身socket *)
    uiErr : UINT;  (* 用于承接功能块中报错引脚错误信息的变量 *)
    isInit : BOOL := FALSE;  (* 用于初始化执行一次的逻辑变量 *)
    arClient : ARRAY[0..10] OF INT;  (* 用于存放Client即主站的socket *)
    btargetAngleChange : BOOL := FALSE;
    OldTargetAngle : WORD;
    enCtr : BOOL := FALSE;  (* Modbus TCP Slave执行功能块使能变量 *)
    iTemp : INT;  (* 临时变量，用于32位数据转换 *)
    dwAngle : INT;  (* 32位临时存储，用于组合角度寄存器 *)
    i : INT;
    wTemp : WORD;  (* modbuslog *)
    sCurLog : STRING(100);
    iLen : INT;
    pCurEntry : POINTER TO LogEntry;
    iCharIdx : INT;
    iRegIdx : INT;
  END_VAR

                    // ================================
// 日志映射部分：将当前未读日志填充到保持寄存器
// ================================
IF g_LogBuffer.count > 0 THEN
    // 获取当前读指针指向的日志条目
    pCurEntry := ADR(g_LogBuffer.entries[g_LogBuffer.readIdx]);
    sCurLog := pCurEntry^.sMessage;
    iLen := pCurEntry^.length;
    
    // 地址100：日志长度（WORD）
    arReg_data[100] := INT_TO_WORD(iLen);
    
    // 地址101-102：时间戳（低字，高字）
    arReg_data[101] := DWORD_TO_WORD(pCurEntry^.timestamp AND 16#FFFF);
    arReg_data[102] := DWORD_TO_WORD(SHR(pCurEntry^.timestamp, 16));
    
    // 清空字符串缓冲区寄存器（地址103 ~ 152，共50个WORD）
    FOR i := 103 TO 152 DO
        arReg_data[i] := 0;
    END_FOR
    
    // ----- 将字符串每两个字符打包成一个 WORD -----
    // 注意：你的环境中字符串索引从0开始（已验证）
    iCharIdx := 0;      // 当前字符索引（从0开始）
    iRegIdx := 103;     // 当前寄存器地址
    WHILE iCharIdx < iLen DO
        // 低字节 = 第一个字符
        wTemp := sCurLog[iCharIdx];
        iCharIdx := iCharIdx + 1;
        // 如果有下一个字符，放入高字节
        IF iCharIdx < iLen THEN
            wTemp := wTemp OR SHL(sCurLog[iCharIdx], 8);
            iCharIdx := iCharIdx + 1;
        END_IF
        arReg_data[iRegIdx] := wTemp;
        iRegIdx := iRegIdx + 1;
    END_WHILE
ELSE
    // 无未读日志，长度寄存器写0
    arReg_data[100] := 0;
END_IF

// --------------------------------
// 处理主站确认线圈（地址16）
// --------------------------------
IF arDo_data[16] THEN
    IF g_LogBuffer.count > 0 THEN
        g_LogBuffer.readIdx := (g_LogBuffer.readIdx + 1) MOD g_LogBuffer.maxSize;
        g_LogBuffer.count := g_LogBuffer.count - 1;
    END_IF
    arDo_data[16] := FALSE;
END_IF



IF isInit=FALSE THEN							

	modtcpslaveinit(en_in:=TRUE,					//Modbus TCP Slave初始化功能块使能
	xenable:=TRUE,									//使能初始化功能
	iport:=502,										//开放端口号502
	en_out=>eout,									//Modbus TCP Slave初始化功能块执行完成
	isocket=>iSocket,								//创建的socket存入变量
	uierror=>uiErr);								//Modbus TCP Slave初始化功能块执行错误信息
	
	IF isocket>=0 AND uiErr=0 THEN					//成功创建socket且无错误，逻辑标志置位，下周期执行ELSE
		isInit:=TRUE;	
		
		enCtr:=FALSE;
		ELSE                                        //等待连接成功
		modtcpslaveinit(en_in:=0,xenable:=0);	
	END_IF
 
ELSE



	// ============================================================
	// v26085 Modbus 寄存器集中处理区
	// 规则：所有 arReg_data/arAi_data 的地址读写都放在本程序，其他程序只写全局缓存变量。
	// ============================================================

	// arAi_data[1..5]：五轴当前位置反馈输入寄存器，X/Y/Z/B/C。
	// Python 按 0.1 单位读取；PLC 内部角度除以 aAngleFactor 后再乘 10。
	FOR i := 1 TO GVL.AXIS_COUNT DO
		arAi_data[i] := INT_TO_WORD(REAL_TO_INT(Axes[i].ActualAngle/aAngleFactor[i]*10.0));
	END_FOR

	// arAi_data[9]：五轴平台运行状态反馈，来自 FiveDOF_Platform_PRG 维护的 bfiveDOF_state。
	arAi_data[9]:=bfiveDOF_state;

	// arReg_data[0]：五轴绝对定位启动命令，非 0 时由 FiveDOF_Platform_PRG 触发运动。
	Move_5Axis_Sign:=arReg_data[0];

	// arReg_data[1..5]：五轴目标位置原始值，只有平台空闲时才更新目标，避免运动中目标被改写。
	IF 	bfiveDOF_state =0 THEN
		FOR i := 1 TO GVL.AXIS_COUNT DO
			dwAngle := WORD_TO_INT(arReg_data[i]);      // 有符号原始值
			PlatformTargetAngle[i] := dwAngle * aAngleFactor[i];
		END_FOR
	END_IF

	// arReg_data[32]：五轴总使能命令。0=关闭使能，非 0=打开使能。
	xEnableAllReg := arReg_data[32] <> 0;
	FOR i := 1 TO GVL.AXIS_COUNT DO
		GVL.Axes[i].AxisEnable := xEnableAllReg;
	END_FOR

	// arReg_data[48]：五轴使能请求反馈，bit0..bit4=X/Y/Z/B/C，bit15=五轴全部请求 TRUE。
	wEnableFeedbackReg := WORD#0;
	IF GVL.Axes[1].AxisEnable THEN wEnableFeedbackReg := wEnableFeedbackReg OR WORD#16#0001; END_IF;
	IF GVL.Axes[2].AxisEnable THEN wEnableFeedbackReg := wEnableFeedbackReg OR WORD#16#0002; END_IF;
	IF GVL.Axes[3].AxisEnable THEN wEnableFeedbackReg := wEnableFeedbackReg OR WORD#16#0004; END_IF;
	IF GVL.Axes[4].AxisEnable THEN wEnableFeedbackReg := wEnableFeedbackReg OR WORD#16#0008; END_IF;
	IF GVL.Axes[5].AxisEnable THEN wEnableFeedbackReg := wEnableFeedbackReg OR WORD#16#0010; END_IF;
	IF GVL.Axes[1].AxisEnable
	   AND GVL.Axes[2].AxisEnable
	   AND GVL.Axes[3].AxisEnable
	   AND GVL.Axes[4].AxisEnable
	   AND GVL.Axes[5].AxisEnable THEN
		wEnableFeedbackReg := wEnableFeedbackReg OR WORD#16#8000;
	END_IF;
	arReg_data[48] := WORD_TO_INT(wEnableFeedbackReg);

	// arReg_data[19]：点动总开关位图，bit0=X，bit1=Y，bit2=Z，bit3=B，bit4=C。
	xJogMode[1] := (arReg_data[19] AND WORD#16#0001) <> WORD#0; // X
	xJogMode[2] := (arReg_data[19] AND WORD#16#0002) <> WORD#0; // Y
	xJogMode[3] := (arReg_data[19] AND WORD#16#0004) <> WORD#0; // Z
	xJogMode[4] := (arReg_data[19] AND WORD#16#0008) <> WORD#0; // B
	xJogMode[5] := (arReg_data[19] AND WORD#16#0010) <> WORD#0; // C

	// arReg_data[6..15]：点动方向命令。方向必须同时满足 arReg_data[19] 对应轴点动总开关。
	xJogFwd[1] := xJogMode[1] AND (arReg_data[6] <> WORD#0);   // X 正向
	xJogRev[1] := xJogMode[1] AND (arReg_data[7] <> WORD#0);   // X 反向
	xJogFwd[2] := xJogMode[2] AND (arReg_data[8] <> WORD#0);   // Y 正向
	xJogRev[2] := xJogMode[2] AND (arReg_data[9] <> WORD#0);   // Y 反向
	xJogFwd[3] := xJogMode[3] AND (arReg_data[10] <> WORD#0);  // Z 正向
	xJogRev[3] := xJogMode[3] AND (arReg_data[11] <> WORD#0);  // Z 反向
	xJogFwd[4] := xJogMode[4] AND (arReg_data[12] <> WORD#0);  // B 正向
	xJogRev[4] := xJogMode[4] AND (arReg_data[13] <> WORD#0);  // B 反向
	xJogFwd[5] := xJogMode[5] AND (arReg_data[14] <> WORD#0);  // C 正向
	xJogRev[5] := xJogMode[5] AND (arReg_data[15] <> WORD#0);  // C 反向

	// arReg_data[89]：五轴复位命令位图，Python 写短脉冲，bit0..bit4=X/Y/Z/B/C。
	xJogReset[1] := (arReg_data[89] AND WORD#16#0001) <> WORD#0; // X 复位
	xJogReset[2] := (arReg_data[89] AND WORD#16#0002) <> WORD#0; // Y 复位
	xJogReset[3] := (arReg_data[89] AND WORD#16#0004) <> WORD#0; // Z 复位
	xJogReset[4] := (arReg_data[89] AND WORD#16#0008) <> WORD#0; // B 复位
	xJogReset[5] := (arReg_data[89] AND WORD#16#0010) <> WORD#0; // C 复位

	// arReg_data[33..37]：五轴状态字，来自 AxisStatusFeedback_PRG 写入的 wAxisStatusReg[1..5]。
	arReg_data[33] := WORD_TO_INT(wAxisStatusReg[1]); // X 状态字
	arReg_data[34] := WORD_TO_INT(wAxisStatusReg[2]); // Y 状态字
	arReg_data[35] := WORD_TO_INT(wAxisStatusReg[3]); // Z 状态字
	arReg_data[36] := WORD_TO_INT(wAxisStatusReg[4]); // B 状态字
	arReg_data[37] := WORD_TO_INT(wAxisStatusReg[5]); // C 状态字

	// arReg_data[38..47]：五轴 AxisErrorID，DWORD 拆成低 16 位和高 16 位。
	arReg_data[38] := WORD_TO_INT(DWORD_TO_WORD(dwAxisErrorIDReg[1]));
arReg_data[39] := WORD_TO_INT(DWORD_TO_WORD(SHR(dwAxisErrorIDReg[1], 16)));
	arReg_data[40] := WORD_TO_INT(DWORD_TO_WORD(dwAxisErrorIDReg[2]));
arReg_data[41] := WORD_TO_INT(DWORD_TO_WORD(SHR(dwAxisErrorIDReg[2], 16)));
	arReg_data[42] := WORD_TO_INT(DWORD_TO_WORD(dwAxisErrorIDReg[3]));
arReg_data[43] := WORD_TO_INT(DWORD_TO_WORD(SHR(dwAxisErrorIDReg[3], 16)));
	arReg_data[44] := WORD_TO_INT(DWORD_TO_WORD(dwAxisErrorIDReg[4]));
arReg_data[45] := WORD_TO_INT(DWORD_TO_WORD(SHR(dwAxisErrorIDReg[4], 16)));
	arReg_data[46] := WORD_TO_INT(DWORD_TO_WORD(dwAxisErrorIDReg[5]));
arReg_data[47] := WORD_TO_INT(DWORD_TO_WORD(SHR(dwAxisErrorIDReg[5], 16)));

	// arReg_data[49..58]：五轴 MC_ReadStatus.ErrorID，DWORD 拆成低 16 位和高 16 位。
	arReg_data[49] := WORD_TO_INT(DWORD_TO_WORD(dwReadStatusErrorIDReg[1]));
arReg_data[50] := WORD_TO_INT(DWORD_TO_WORD(SHR(dwReadStatusErrorIDReg[1], 16)));
	arReg_data[51] := WORD_TO_INT(DWORD_TO_WORD(dwReadStatusErrorIDReg[2]));
arReg_data[52] := WORD_TO_INT(DWORD_TO_WORD(SHR(dwReadStatusErrorIDReg[2], 16)));
	arReg_data[53] := WORD_TO_INT(DWORD_TO_WORD(dwReadStatusErrorIDReg[3]));
arReg_data[54] := WORD_TO_INT(DWORD_TO_WORD(SHR(dwReadStatusErrorIDReg[3], 16)));
	arReg_data[55] := WORD_TO_INT(DWORD_TO_WORD(dwReadStatusErrorIDReg[4]));
arReg_data[56] := WORD_TO_INT(DWORD_TO_WORD(SHR(dwReadStatusErrorIDReg[4], 16)));
	arReg_data[57] := WORD_TO_INT(DWORD_TO_WORD(dwReadStatusErrorIDReg[5]));
arReg_data[58] := WORD_TO_INT(DWORD_TO_WORD(SHR(dwReadStatusErrorIDReg[5], 16)));

	// arReg_data[59..68]：五轴 MC_ReadAxisError.ErrorID，DWORD 拆成低 16 位和高 16 位。
	arReg_data[59] := WORD_TO_INT(DWORD_TO_WORD(dwReadAxisErrorFBIDReg[1]));
arReg_data[60] := WORD_TO_INT(DWORD_TO_WORD(SHR(dwReadAxisErrorFBIDReg[1], 16)));
	arReg_data[61] := WORD_TO_INT(DWORD_TO_WORD(dwReadAxisErrorFBIDReg[2]));
arReg_data[62] := WORD_TO_INT(DWORD_TO_WORD(SHR(dwReadAxisErrorFBIDReg[2], 16)));
	arReg_data[63] := WORD_TO_INT(DWORD_TO_WORD(dwReadAxisErrorFBIDReg[3]));
arReg_data[64] := WORD_TO_INT(DWORD_TO_WORD(SHR(dwReadAxisErrorFBIDReg[3], 16)));
	arReg_data[65] := WORD_TO_INT(DWORD_TO_WORD(dwReadAxisErrorFBIDReg[4]));
arReg_data[66] := WORD_TO_INT(DWORD_TO_WORD(SHR(dwReadAxisErrorFBIDReg[4], 16)));
	arReg_data[67] := WORD_TO_INT(DWORD_TO_WORD(dwReadAxisErrorFBIDReg[5]));
arReg_data[68] := WORD_TO_INT(DWORD_TO_WORD(SHR(dwReadAxisErrorFBIDReg[5], 16)));

	// arReg_data[69..78]：五轴 MC_Power.ErrorID，DWORD 拆成低 16 位和高 16 位。
	arReg_data[69] := WORD_TO_INT(DWORD_TO_WORD(dwPowerErrorIDReg[1]));
arReg_data[70] := WORD_TO_INT(DWORD_TO_WORD(SHR(dwPowerErrorIDReg[1], 16)));
	arReg_data[71] := WORD_TO_INT(DWORD_TO_WORD(dwPowerErrorIDReg[2]));
arReg_data[72] := WORD_TO_INT(DWORD_TO_WORD(SHR(dwPowerErrorIDReg[2], 16)));
	arReg_data[73] := WORD_TO_INT(DWORD_TO_WORD(dwPowerErrorIDReg[3]));
arReg_data[74] := WORD_TO_INT(DWORD_TO_WORD(SHR(dwPowerErrorIDReg[3], 16)));
	arReg_data[75] := WORD_TO_INT(DWORD_TO_WORD(dwPowerErrorIDReg[4]));
arReg_data[76] := WORD_TO_INT(DWORD_TO_WORD(SHR(dwPowerErrorIDReg[4], 16)));
	arReg_data[77] := WORD_TO_INT(DWORD_TO_WORD(dwPowerErrorIDReg[5]));
arReg_data[78] := WORD_TO_INT(DWORD_TO_WORD(SHR(dwPowerErrorIDReg[5], 16)));

	// arReg_data[79..83]：五轴 MC_Power 诊断字，bit0=Status，bit1=Error。
	arReg_data[79] := WORD_TO_INT(wPowerDiagReg[1]); // X MC_Power 诊断
	arReg_data[80] := WORD_TO_INT(wPowerDiagReg[2]); // Y MC_Power 诊断
	arReg_data[81] := WORD_TO_INT(wPowerDiagReg[3]); // Z MC_Power 诊断
	arReg_data[82] := WORD_TO_INT(wPowerDiagReg[4]); // B MC_Power 诊断
	arReg_data[83] := WORD_TO_INT(wPowerDiagReg[5]); // C MC_Power 诊断

	// arReg_data[84..88]：轴状态诊断版本和汇总位图。
	arReg_data[84] := 26085;                              // 诊断版本号
	arReg_data[85] := WORD_TO_INT(wEnableMismatchReg);        // 使能请求不一致位图
	arReg_data[86] := WORD_TO_INT(wReadStatusErrorBitsReg);   // MC_ReadStatus.Error 位图
	arReg_data[87] := WORD_TO_INT(wReadAxisErrorBitsReg);     // MC_ReadAxisError.Error 位图
	arReg_data[88] := WORD_TO_INT(wReadStatusFBErrorBitsReg); // MC_ReadStatus.FBErrorOccured 位图

	// arReg_data[90..99]：点动/复位诊断反馈，全部由 Jog 程序写全局缓存，本程序统一输出到 Modbus。
	arReg_data[90] := WORD_TO_INT(wJogResetCmdReg); // 复位命令读到反馈
	arReg_data[91] := WORD_TO_INT(wJogModeReg);     // 点动总开关反馈
	arReg_data[92] := WORD_TO_INT(wJogFwdReg);      // 正向点动命令反馈
	arReg_data[93] := WORD_TO_INT(wJogRevReg);      // 反向点动命令反馈
	arReg_data[94] := WORD_TO_INT(wJogReadyReg);    // FB_ServoJog.xReady
	arReg_data[95] := WORD_TO_INT(wJogMovingReg);   // FB_ServoJog.xMoving
	arReg_data[96] := WORD_TO_INT(wJogFaultReg);    // FB_ServoJog.xFault
	arReg_data[97] := WORD_TO_INT(wJogErrorReg);    // FB_ServoJog.xJogError
	arReg_data[98] := WORD_TO_INT(wJogAbortedReg);  // FB_ServoJog.xJogAborted
	arReg_data[99] := 26085;                    // 点动/复位诊断版本号
	modtcpslavectrl(en_in:=enCtr,					//Modbus TCP Slave执行功能块使能
	xenable:=TRUE,									//Modbus TCP Slave执行功能使能
	isocket:=isocket,								//输入创建的socket
	dwatchdogtime:=2000,							//看门狗时间
	p_clientsocket:=ADR(arClient),					//将连接进来的socket存放到数组
	imaxclientcount:=10,							//设置最大连接数量
	uido_number:=17,uido_startaddr:=0,pdo_data:=ADR(arDo_data),		//uido_number设定线圈个数，uido_startaddr设定线圈起始地址，数据存放在arDo_data数组
	uidi_number:=16,uidi_startaddr:=0,pdi_data:=ADR(arDi_data),		//uidi_number设定离散型数据个数，uidi_startaddr设定离散型数据起始地址，数据存放在arDi_data数组
	uireg_number:=200,uireg_startaddr:=0,preg_data:=ADR(arReg_data), //uireg_number设定保持型寄存器个数，uireg_startaddr设定保持型寄存器起始地址，数据存放在arReg_data数组
	uiai_number:=16,uiai_startaddr:=0,pai_data:=ADR(arAi_data),		//uiai_number设定输入型寄存器个数，uiai_startaddr设定输入型寄存器起始地址，数据存放在arAi_data数组
	en_out=>eout,									//Modbus TCP Slave执行功能块执行完成
	uierror=>uierr);								//Modbus TCP Slave执行功能块执行错误信息
	enctr:=TRUE;
	IF uierr <>0 THEN                               //如果从站报错，则重新连接从站
		modtcpslaveinit(en_in:=0,xenable:=0);	
		isInit:=0;
	END_IF
END_IF

 
// 释放锁
g_LogLock := FALSE;
 
                  
END_PROGRAM

CONFIGURATION Device
  RESOURCE Application ON PLC
    VAR_GLOBAL CONSTANT  (* GVL *)
      AXIS_COUNT : INT := 5;
      使能 : BOOL;  (* 接收到的目标角度（浮点数） *)
      Axes : ARRAY[1..5] OF Axis;  (* 5个轴的结构体数组 *)
      Move_5Axis_Sign : INT;
      step : INT := 0;  (* 0空闲, 10平台运动 20运动完成 *)
      bModeSwitchDone : BOOL := FALSE;
      torque_pos_change : BOOL := TRUE;
      PlatformTargetAngle : ARRAY[1..AXIS_COUNT] OF LREAL;
      PlatformTargetVel : ARRAY[1..AXIS_COUNT] OF LREAL;
      pushmotorpos : LREAL;
      arDo_data : ARRAY[0..16] OF BOOL;  (* 用于存放线圈的数据 *)
      arDi_data : ARRAY[0..15] OF BOOL;  (* 用于存放离散型数据 *)
      arReg_data : ARRAY[0..199] OF INT;  (* 用于存放保持型寄存器的数据 *)
      arAi_data : ARRAY[0..16] OF INT;  (* 用于存放输入型寄存器的数据 *)
      mchome : Sm3_Basic.MC_Home;
      DoorlockHomedone : BOOL;
      StrikeplateHomedone : BOOL;
      bfiveDOF_state : INT;
      xJogFwd : ARRAY[1..5] OF BOOL;
      xJogRev : ARRAY[1..5] OF BOOL;
      xJogMode : ARRAY[1..5] OF BOOL;
      g_LogBuffer : LogBuffer := (writeIdx := 0, readIdx := 0, count := 0, maxSize := 10);  (* 日志modbus 日志缓冲区配置 *)
      g_bLogNew : BOOL;  (* 可选：有新日志标志（供主站快速判断） *)
      g_LogLock : BOOL := FALSE;  (* 互斥标志 *)
      g_LogQueue : ARRAY[0..199] OF LogQueueEntry;  (* 增大队列深度 *)
      g_QueueHead : INT := 0;
      g_QueueTail : INT := 0;
      g_QueueCount : INT := 0;
      g_QueueLock : BOOL := FALSE;
      xJogReset : ARRAY[1..5] OF BOOL;
      wAxisStatusReg : ARRAY[1..5] OF WORD;
      dwAxisErrorIDReg : ARRAY[1..5] OF DWORD;
      dwReadStatusErrorIDReg : ARRAY[1..5] OF DWORD;
      dwReadAxisErrorFBIDReg : ARRAY[1..5] OF DWORD;
      dwPowerErrorIDReg : ARRAY[1..5] OF DWORD;
      wPowerDiagReg : ARRAY[1..5] OF WORD;
      wEnableFeedbackReg : WORD;
      wEnableMismatchReg : WORD;
      wReadStatusErrorBitsReg : WORD;
      wReadAxisErrorBitsReg : WORD;
      wReadStatusFBErrorBitsReg : WORD;
      wJogResetCmdReg : WORD;
      wJogModeReg : WORD;
      wJogFwdReg : WORD;
      wJogRevReg : WORD;
      wJogReadyReg : WORD;
      wJogMovingReg : WORD;
      wJogFaultReg : WORD;
      wJogErrorReg : WORD;
      wJogAbortedReg : WORD;
    END_VAR
  END_RESOURCE
END_CONFIGURATION
